// TwinCAT 3 PLC project PLC_Project_XYZ
// ProgramVersion: 3.1.4026.12
// CompilerDefines: VISU_USEPROPERTYINFO
// libraries:
//   Tc2_MC2, * (Beckhoff Automation GmbH)
//   Tc2_Standard, * (Beckhoff Automation GmbH)
//   Tc2_System, * (Beckhoff Automation GmbH)
//   Tc3_Module, * (Beckhoff Automation GmbH)
//   VisuSymbols, 4.5.0.0 (System)
// project tree:
//   / GlobalTextList.TcGTLO, PlcTask.TcTTO, Visualization Manager.TcVMO (not stored)
//   GVLs/ GVL.TcGVL
//   POUs/ MAIN.TcPOU
//   VISUs/ Visu.TcVIS
// real-time tasks:
//   TASK PlcTask: cycle T#10ms, priority 20, ADS port 350
// motion (NC):
//   TASK NC-Task 1 SAF: cycle T#2ms, priority 4, ADS port 501
//   TASK NC-Task 1 SVB: cycle T#10ms, priority 8, ADS port 511
//   AXIS Axis 1 (id 1)
//     OtherSettings: AllowMotionCmdToSlave=true
//     encoder EncType=4
//       EncPara: ScaleFactorNumerator=60, ScaleFactorDenominator=12800, MaxCount=#x0000ffff
//         Inc: RefSoftSyncMask=#x0000ffff
//     drive DrvType=24
//       Analog: VeloReferenz=600, TorqueSetpointScale=10, ScaleFactorActTorque=0.1
//       TimeComp: TaskDelayCycles=1
//     controller CtrType=1
//       CtrPara: PriorControlFactor=1
//         Observer: BandWidth=20
//   AXIS Axis 2 (id 2)
//     OtherSettings: AllowMotionCmdToSlave=true
//     encoder EncType=4
//       EncPara: ScaleFactorNumerator=60, ScaleFactorDenominator=12800, MaxCount=#x0000ffff
//         Inc: RefSoftSyncMask=#x0000ffff
//     drive DrvType=24
//       Analog: VeloReferenz=600, TorqueSetpointScale=10, ScaleFactorActTorque=0.1
//       TimeComp: TaskDelayCycles=1
//     controller CtrType=1
//       CtrPara: PriorControlFactor=1
//         Observer: BandWidth=20
//   AXIS Axis 3 (id 3)
//     OtherSettings: AllowMotionCmdToSlave=true
//     encoder EncType=4
//       EncPara: ScaleFactorNumerator=60, ScaleFactorDenominator=12800, MaxCount=#x0000ffff
//         Inc: RefSoftSyncMask=#x0000ffff
//     drive DrvType=24
//       Analog: VeloReferenz=600, TorqueSetpointScale=10, ScaleFactorActTorque=0.1
//       TimeComp: TaskDelayCycles=1
//     controller CtrType=1
//       CtrPara: PriorControlFactor=1
//         Observer: BandWidth=20
//   AXIS Axis 4 (id 4)
//     OtherSettings: AllowMotionCmdToSlave=true
//     encoder EncType=4
//       EncPara: ScaleFactorNumerator=60, ScaleFactorDenominator=12800, MaxCount=#x0000ffff
//         Inc: RefSoftSyncMask=#x0000ffff
//     drive DrvType=24
//       Analog: VeloReferenz=600, TorqueSetpointScale=10, ScaleFactorActTorque=0.1
//       TimeComp: TaskDelayCycles=1
//     controller CtrType=1
//       CtrPara: PriorControlFactor=1
//         Observer: BandWidth=20
// I/O:
//   DEVICE Device 1 (EtherCAT), AmsNetId 199.4.42.250.2.1
//     Term 1 (EK1200) [EK1200-5000 EtherCAT Power supply (2A E-Bus)]
//       Term 2 (EL1008) [EL1008 8Ch. Dig. Input 24V, 3ms]
//       Term 3 (EL2008) [EL2008 8Ch. Dig. Output 24V, 0.5A]
//       Term 4 (EL3062) [EL3062 2Ch. Ana. Input 0-10V]
//       Term 5 (EL4002) [EL4002 2Ch. Ana. Output 0-10V, 12bit]
//       Term 6 (EK1110) [EK1110 EtherCAT extension]
//     Term 7 (EK1100) [EK1100 EtherCAT Coupler (2A E-Bus)]
//       Term 8 (EL7031-0030) [EL7031-0030 1Ch. Stepper motor output stage (24V, 2.8A)]
//       Term 9 (EL7031-0030) [EL7031-0030 1Ch. Stepper motor output stage (24V, 2.8A)]
//       Term 10 (EL7031-0030) [EL7031-0030 1Ch. Stepper motor output stage (24V, 2.8A)]
//       Term 11 (EL7031-0030) [EL7031-0030 1Ch. Stepper motor output stage (24V, 2.8A)]
//       Term 12 (EL1008) [EL1008 8Ch. Dig. Input 24V, 3ms]
//       Term 13 (EK1110) [EK1110 EtherCAT extension]
//   DEVICE Device 2 (EtherCAT Automation Protocol), AmsNetId 199.4.42.250.3.1
//   DEVICE Device 3 (NOV-DP-RAM)
// variable links:
//   NC-Task 1 SAF/Axes/Axis 1 <-> Device 1 (EtherCAT)/Term 7 (EK1100)/Term 8 (EL7031-0030)
//     Drive/Inputs/In/nState1 @bit 3 <-> STM Status/Status/Error
//     Drive/Inputs/In/nState1 @bit 5 <-> STM Status/Status/Moving negative
//     Drive/Inputs/In/nState1 @bit 4 <-> STM Status/Status/Moving positive
//     Drive/Inputs/In/nState1 @bit 1 <-> STM Status/Status/Ready
//     Drive/Inputs/In/nState1 <-> STM Status/Status/Ready to enable
//     Drive/Inputs/In/nState1 @bit 6 <-> STM Status/Status/Torque reduced
//     Drive/Inputs/In/nState1 @bit 2 <-> STM Status/Status/Warning
//     Drive/Inputs/In/nState2 @bit 3 <-> STM Status/Status/Digital input 1
//     Drive/Inputs/In/nState2 @bit 4 <-> STM Status/Status/Digital input 2
//     Drive/Inputs/In/nState2 @bit 5 <-> STM Status/Status/Sync error
//     Drive/Inputs/In/nState2 @bit 7 <-> STM Status/Status/TxPDO Toggle
//     Drive/Inputs/In/nState4 @bit 1 <-> WcState/InputToggle
//     Drive/Inputs/In/nState4 <-> WcState/WcState
//     Drive/Outputs/Out/nCtrl1 <-> STM Control/Control/Enable
//     Drive/Outputs/Out/nCtrl1 @bit 2 <-> STM Control/Control/Reduce torque
//     Drive/Outputs/Out/nCtrl1 @bit 1 <-> STM Control/Control/Reset
//     Drive/Outputs/Out/nDataOut2[0] <-> STM Velocity/Velocity
//     Enc/Inputs/In/nDataIn1[0] <-> ENC Status compact/Counter value
//     Enc/Inputs/In/nDataIn2[0] <-> ENC Status compact/Latch value
//     Enc/Inputs/In/nState1 @bit 4 <-> ENC Status compact/Status/Counter overflow
//     Enc/Inputs/In/nState1 @bit 3 <-> ENC Status compact/Status/Counter underflow
//     Enc/Inputs/In/nState1 @bit 1 <-> ENC Status compact/Status/Latch extern valid
//     Enc/Inputs/In/nState1 @bit 2 <-> ENC Status compact/Status/Set counter done
//     Enc/Inputs/In/nState2 @bit 4 <-> ENC Status compact/Status/Status of extern latch
//     Enc/Inputs/In/nState2 @bit 5 <-> ENC Status compact/Status/Sync error
//     Enc/Inputs/In/nState2 @bit 7 <-> ENC Status compact/Status/TxPDO Toggle
//     Enc/Inputs/In/nState4 @bit 1 <-> WcState/InputToggle
//     Enc/Inputs/In/nState4 <-> WcState/WcState
//     Enc/Outputs/Out/nCtrl1 @bit 3 <-> ENC Control compact/Control/Enable latch extern on negative edge
//     Enc/Outputs/Out/nCtrl1 @bit 1 <-> ENC Control compact/Control/Enable latch extern on positive edge
//     Enc/Outputs/Out/nCtrl1 @bit 2 <-> ENC Control compact/Control/Set counter
//     Enc/Outputs/Out/nDataOut1[0] <-> ENC Control compact/Set counter value
//   NC-Task 1 SAF/Axes/Axis 2 <-> Device 1 (EtherCAT)/Term 7 (EK1100)/Term 9 (EL7031-0030)
//     Drive/Inputs/In/nState1 @bit 3 <-> STM Status/Status/Error
//     Drive/Inputs/In/nState1 @bit 5 <-> STM Status/Status/Moving negative
//     Drive/Inputs/In/nState1 @bit 4 <-> STM Status/Status/Moving positive
//     Drive/Inputs/In/nState1 @bit 1 <-> STM Status/Status/Ready
//     Drive/Inputs/In/nState1 <-> STM Status/Status/Ready to enable
//     Drive/Inputs/In/nState1 @bit 6 <-> STM Status/Status/Torque reduced
//     Drive/Inputs/In/nState1 @bit 2 <-> STM Status/Status/Warning
//     Drive/Inputs/In/nState2 @bit 3 <-> STM Status/Status/Digital input 1
//     Drive/Inputs/In/nState2 @bit 4 <-> STM Status/Status/Digital input 2
//     Drive/Inputs/In/nState2 @bit 5 <-> STM Status/Status/Sync error
//     Drive/Inputs/In/nState2 @bit 7 <-> STM Status/Status/TxPDO Toggle
//     Drive/Inputs/In/nState4 @bit 1 <-> WcState/InputToggle
//     Drive/Inputs/In/nState4 <-> WcState/WcState
//     Drive/Outputs/Out/nCtrl1 <-> STM Control/Control/Enable
//     Drive/Outputs/Out/nCtrl1 @bit 2 <-> STM Control/Control/Reduce torque
//     Drive/Outputs/Out/nCtrl1 @bit 1 <-> STM Control/Control/Reset
//     Drive/Outputs/Out/nDataOut2[0] <-> STM Velocity/Velocity
//     Enc/Inputs/In/nDataIn1[0] <-> ENC Status compact/Counter value
//     Enc/Inputs/In/nDataIn2[0] <-> ENC Status compact/Latch value
//     Enc/Inputs/In/nState1 @bit 4 <-> ENC Status compact/Status/Counter overflow
//     Enc/Inputs/In/nState1 @bit 3 <-> ENC Status compact/Status/Counter underflow
//     Enc/Inputs/In/nState1 @bit 1 <-> ENC Status compact/Status/Latch extern valid
//     Enc/Inputs/In/nState1 @bit 2 <-> ENC Status compact/Status/Set counter done
//     Enc/Inputs/In/nState2 @bit 4 <-> ENC Status compact/Status/Status of extern latch
//     Enc/Inputs/In/nState2 @bit 5 <-> ENC Status compact/Status/Sync error
//     Enc/Inputs/In/nState2 @bit 7 <-> ENC Status compact/Status/TxPDO Toggle
//     Enc/Inputs/In/nState4 @bit 1 <-> WcState/InputToggle
//     Enc/Inputs/In/nState4 <-> WcState/WcState
//     Enc/Outputs/Out/nCtrl1 @bit 3 <-> ENC Control compact/Control/Enable latch extern on negative edge
//     Enc/Outputs/Out/nCtrl1 @bit 1 <-> ENC Control compact/Control/Enable latch extern on positive edge
//     Enc/Outputs/Out/nCtrl1 @bit 2 <-> ENC Control compact/Control/Set counter
//     Enc/Outputs/Out/nDataOut1[0] <-> ENC Control compact/Set counter value
//   NC-Task 1 SAF/Axes/Axis 3 <-> Device 1 (EtherCAT)/Term 7 (EK1100)/Term 10 (EL7031-0030)
//     Drive/Inputs/In/nState1 @bit 3 <-> STM Status/Status/Error
//     Drive/Inputs/In/nState1 @bit 5 <-> STM Status/Status/Moving negative
//     Drive/Inputs/In/nState1 @bit 4 <-> STM Status/Status/Moving positive
//     Drive/Inputs/In/nState1 @bit 1 <-> STM Status/Status/Ready
//     Drive/Inputs/In/nState1 <-> STM Status/Status/Ready to enable
//     Drive/Inputs/In/nState1 @bit 6 <-> STM Status/Status/Torque reduced
//     Drive/Inputs/In/nState1 @bit 2 <-> STM Status/Status/Warning
//     Drive/Inputs/In/nState2 @bit 3 <-> STM Status/Status/Digital input 1
//     Drive/Inputs/In/nState2 @bit 4 <-> STM Status/Status/Digital input 2
//     Drive/Inputs/In/nState2 @bit 5 <-> STM Status/Status/Sync error
//     Drive/Inputs/In/nState2 @bit 7 <-> STM Status/Status/TxPDO Toggle
//     Drive/Inputs/In/nState4 @bit 1 <-> WcState/InputToggle
//     Drive/Inputs/In/nState4 <-> WcState/WcState
//     Drive/Outputs/Out/nCtrl1 <-> STM Control/Control/Enable
//     Drive/Outputs/Out/nCtrl1 @bit 2 <-> STM Control/Control/Reduce torque
//     Drive/Outputs/Out/nCtrl1 @bit 1 <-> STM Control/Control/Reset
//     Drive/Outputs/Out/nDataOut2[0] <-> STM Velocity/Velocity
//     Enc/Inputs/In/nDataIn1[0] <-> ENC Status compact/Counter value
//     Enc/Inputs/In/nDataIn2[0] <-> ENC Status compact/Latch value
//     Enc/Inputs/In/nState1 @bit 4 <-> ENC Status compact/Status/Counter overflow
//     Enc/Inputs/In/nState1 @bit 3 <-> ENC Status compact/Status/Counter underflow
//     Enc/Inputs/In/nState1 @bit 1 <-> ENC Status compact/Status/Latch extern valid
//     Enc/Inputs/In/nState1 @bit 2 <-> ENC Status compact/Status/Set counter done
//     Enc/Inputs/In/nState2 @bit 4 <-> ENC Status compact/Status/Status of extern latch
//     Enc/Inputs/In/nState2 @bit 5 <-> ENC Status compact/Status/Sync error
//     Enc/Inputs/In/nState2 @bit 7 <-> ENC Status compact/Status/TxPDO Toggle
//     Enc/Inputs/In/nState4 @bit 1 <-> WcState/InputToggle
//     Enc/Inputs/In/nState4 <-> WcState/WcState
//     Enc/Outputs/Out/nCtrl1 @bit 3 <-> ENC Control compact/Control/Enable latch extern on negative edge
//     Enc/Outputs/Out/nCtrl1 @bit 1 <-> ENC Control compact/Control/Enable latch extern on positive edge
//     Enc/Outputs/Out/nCtrl1 @bit 2 <-> ENC Control compact/Control/Set counter
//     Enc/Outputs/Out/nDataOut1[0] <-> ENC Control compact/Set counter value
//   NC-Task 1 SAF/Axes/Axis 4 <-> Device 1 (EtherCAT)/Term 7 (EK1100)/Term 11 (EL7031-0030)
//     Drive/Inputs/In/nState1 @bit 3 <-> STM Status/Status/Error
//     Drive/Inputs/In/nState1 @bit 5 <-> STM Status/Status/Moving negative
//     Drive/Inputs/In/nState1 @bit 4 <-> STM Status/Status/Moving positive
//     Drive/Inputs/In/nState1 @bit 1 <-> STM Status/Status/Ready
//     Drive/Inputs/In/nState1 <-> STM Status/Status/Ready to enable
//     Drive/Inputs/In/nState1 @bit 6 <-> STM Status/Status/Torque reduced
//     Drive/Inputs/In/nState1 @bit 2 <-> STM Status/Status/Warning
//     Drive/Inputs/In/nState2 @bit 3 <-> STM Status/Status/Digital input 1
//     Drive/Inputs/In/nState2 @bit 4 <-> STM Status/Status/Digital input 2
//     Drive/Inputs/In/nState2 @bit 5 <-> STM Status/Status/Sync error
//     Drive/Inputs/In/nState2 @bit 7 <-> STM Status/Status/TxPDO Toggle
//     Drive/Inputs/In/nState4 @bit 1 <-> WcState/InputToggle
//     Drive/Inputs/In/nState4 <-> WcState/WcState
//     Drive/Outputs/Out/nCtrl1 <-> STM Control/Control/Enable
//     Drive/Outputs/Out/nCtrl1 @bit 2 <-> STM Control/Control/Reduce torque
//     Drive/Outputs/Out/nCtrl1 @bit 1 <-> STM Control/Control/Reset
//     Drive/Outputs/Out/nDataOut2[0] <-> STM Velocity/Velocity
//     Enc/Inputs/In/nDataIn1[0] <-> ENC Status compact/Counter value
//     Enc/Inputs/In/nDataIn2[0] <-> ENC Status compact/Latch value
//     Enc/Inputs/In/nState1 @bit 4 <-> ENC Status compact/Status/Counter overflow
//     Enc/Inputs/In/nState1 @bit 3 <-> ENC Status compact/Status/Counter underflow
//     Enc/Inputs/In/nState1 @bit 1 <-> ENC Status compact/Status/Latch extern valid
//     Enc/Inputs/In/nState1 @bit 2 <-> ENC Status compact/Status/Set counter done
//     Enc/Inputs/In/nState2 @bit 4 <-> ENC Status compact/Status/Status of extern latch
//     Enc/Inputs/In/nState2 @bit 5 <-> ENC Status compact/Status/Sync error
//     Enc/Inputs/In/nState2 @bit 7 <-> ENC Status compact/Status/TxPDO Toggle
//     Enc/Inputs/In/nState4 @bit 1 <-> WcState/InputToggle
//     Enc/Inputs/In/nState4 <-> WcState/WcState
//     Enc/Outputs/Out/nCtrl1 @bit 3 <-> ENC Control compact/Control/Enable latch extern on negative edge
//     Enc/Outputs/Out/nCtrl1 @bit 1 <-> ENC Control compact/Control/Enable latch extern on positive edge
//     Enc/Outputs/Out/nCtrl1 @bit 2 <-> ENC Control compact/Control/Set counter
//     Enc/Outputs/Out/nDataOut1[0] <-> ENC Control compact/Set counter value
//   PLC_Project_XYZ/PLC_Project_XYZ Instance <-> Device 1 (EtherCAT)/Term 1 (EK1200)/Term 2 (EL1008)
//     PlcTask Inputs/MAIN.BTN_LEFT <-> Channel 1/Input
//     PlcTask Inputs/MAIN.BTN_LEFT_B <-> Channel 3/Input
//     PlcTask Inputs/MAIN.BTN_RIGHT <-> Channel 2/Input
//     PlcTask Inputs/MAIN.BTN_RIGHT_B <-> Channel 4/Input
//   PLC_Project_XYZ/PLC_Project_XYZ Instance <-> Device 1 (EtherCAT)/Term 1 (EK1200)/Term 4 (EL3062)
//     PlcTask Inputs/MAIN.nPotentiometer <-> AI Standard Channel 1/Value
//   PLC_Project_XYZ/PLC_Project_XYZ Instance <-> Device 1 (EtherCAT)/Term 7 (EK1100)/Term 12 (EL1008)
//     PlcTask Inputs/MAIN.SWX1 <-> Channel 2/Input
//     PlcTask Inputs/MAIN.SWX2 <-> Channel 1/Input
//     PlcTask Inputs/MAIN.SWY1 <-> Channel 3/Input
//     PlcTask Inputs/MAIN.SWY2 <-> Channel 4/Input
//   PLC_Project_XYZ/PLC_Project_XYZ Instance <-> NC-Task 1 SAF/Axes/Axis 1
//     PlcTask Inputs/MAIN.Axis_y1.NcToPlc <-> Outputs/ToPlc
//     PlcTask Outputs/MAIN.Axis_y1.PlcToNc <-> Inputs/FromPlc
//   PLC_Project_XYZ/PLC_Project_XYZ Instance <-> NC-Task 1 SAF/Axes/Axis 2
//     PlcTask Inputs/MAIN.Axis_y2.NcToPlc <-> Outputs/ToPlc
//     PlcTask Outputs/MAIN.Axis_y2.PlcToNc <-> Inputs/FromPlc
//   PLC_Project_XYZ/PLC_Project_XYZ Instance <-> NC-Task 1 SAF/Axes/Axis 3
//     PlcTask Inputs/MAIN.Axis_z.NcToPlc <-> Outputs/ToPlc
//     PlcTask Outputs/MAIN.Axis_z.PlcToNc <-> Inputs/FromPlc
//   PLC_Project_XYZ/PLC_Project_XYZ Instance <-> NC-Task 1 SAF/Axes/Axis 4
//     PlcTask Inputs/MAIN.Axis_x.NcToPlc <-> Outputs/ToPlc
//     PlcTask Outputs/MAIN.Axis_x.PlcToNc <-> Inputs/FromPlc

CONFIGURATION PLC_Project_XYZ
    RESOURCE PLC ON TwinCAT3
        TASK PlcTask(INTERVAL := T#10ms, PRIORITY := 20);
        PROGRAM MAIN WITH PlcTask : MAIN;
    END_RESOURCE
END_CONFIGURATION

// ---- GVLs/GVL.TcGVL
{attribute 'qualified_only'}
VAR_GLOBAL
	//Leds
	bLed_Rd1 AT %Q* : BOOL;
	bLed_Rd2 AT %Q* : BOOL;
	bLed_Rd3 AT %Q* : BOOL;
	bLed_Rd4 AT %Q* : BOOL;
	
	bLed_Gn1 AT %Q* : BOOL;
	bLed_Gn2 AT %Q* : BOOL;
	bLed_Gn3 AT %Q* : BOOL;
	bLed_Gn4 AT %Q* : BOOL;
	
	//Buttons
	bButton1 	AT %I* : BOOL;
    bButton2 	AT %I* : BOOL;
    bButton3 	AT %I* : BOOL;
    bButton4 	AT %I* : BOOL;
	bButton5 	AT %I* : BOOL;
    bButton6 	AT %I* : BOOL;
	bHome 		AT %I* : BOOL;
	
	//Sliders
	slider1 : INT;
	slider2 : INT;
	slider3 : INT;
END_VAR

// ---- POUs/MAIN.TcPOU
PROGRAM MAIN
VAR

	START : BOOL := FALSE;

    // input
	bJogF	: BOOL := FALSE;
	bJogB	: BOOL := FALSE;
	bSet 	: BOOL := FALSE;
	bToggle : BOOL := FALSE;
	nValue AT %I*: LREAL;
    nPotentiometer AT %I*: INT;
    nDisplay AT %Q*: INT;
	
	
    ExecuteABS        : BOOL;
    Enable          : BOOL := TRUE;
    Enable_Positive : BOOL := TRUE;
    Enable_Negative : BOOL := TRUE;
    Override        : LREAL := 100.0;
    BufferMode      : MC_BufferMode;
    Options         : ST_PowerOptions;
    BTN_RIGHT       AT %I* : BOOL := FALSE;
    BTN_LEFT        AT %I* : BOOL := FALSE;

	BTN_RIGHT_B		AT %I* : BOOL := FALSE;
	BTN_LEFT_B		AT %I* : BOOL := FALSE;
	
    SWY1  AT %I* : BOOL;
    SWY2  AT %I* : BOOL;
    SWX1  AT %I* : BOOL;
    SWX2  AT %I* : BOOL;

    // output
    Status  : BOOL;
    Busy    : BOOL;
    Active  : BOOL;
    Error   : BOOL;
    ErrorID : UDINT;



	



    Axis_x : AXIS_REF;
	Axis_z : AXIS_REF;
	
	Axis_y1 : AXIS_REF;
	Axis_y2 : AXIS_REF;
	
	

    mc_power : MC_Power;
	mc_powerZ : MC_Power;
	mc_powerY1: MC_Power;
	mc_powerY2: MC_Power;

    fbMoveAbsX1: MC_MoveAbsolute;
    fbMoveAbsX2: MC_MoveAbsolute;
	fbMoveAbsY1: MC_MoveAbsolute;
    fbMoveAbsY2: MC_MoveAbsolute;
	fbMoveAbsZ1: MC_MoveAbsolute;
    fbMoveAbsZ2: MC_MoveAbsolute;
	

	Axis_x_Halt: MC_Halt;
	Halt_X1: MC_Halt;
	Halt_X2: MC_Halt;
	
	Axis_y_Halt: MC_Halt;
	Halt_Y1: MC_Halt;
	Halt_Y2: MC_Halt;
	
	Axis_z_Halt: MC_Halt;
	Halt_Z1: MC_Halt;
	Halt_Z2: MC_Halt;
	
	
	Couple_Y1_Y2: MC_GearInDyn;
	fb_Jog_Z: MC_Jog;
	fb_Jog_X: MC_Jog;
	fb_Jog_Y: MC_Jog;
	
END_VAR

mc_power.Enable := Enable;
mc_powerZ.Enable := Enable;
mc_powerY1.Enable:= Enable;
mc_powerY2.Enable:= Enable;

mc_power.Enable_Positive := Enable_Positive;
mc_power.Enable_Negative := Enable_Negative;
mc_power.Override := Override;

mc_powerZ.Enable_Positive := Enable_Positive;
mc_powerZ.Enable_Negative := Enable_Negative;
mc_powerZ.Override := Override;

mc_powerY1.Enable_Positive := Enable_Positive;
mc_powerY1.Enable_Negative := Enable_Negative;
mc_powerY1.Override := Override;

mc_powerY2.Enable_Positive := Enable_Positive;
mc_powerY2.Enable_Negative := Enable_Negative;
mc_powerY2.Override := Override;

mc_power(Axis := Axis_x );
mc_powerZ(Axis := Axis_z );
mc_powerY1(Axis := Axis_y1 );
mc_powerY2(Axis := Axis_y2 );


Couple_Y1_Y2(
	Master:= Axis_y1, 
	Slave:= Axis_y2, 
	Enable:= TRUE, 
	GearRatio:= 1, 
	Acceleration:= , 
	Deceleration:= , 
	Jerk:= , 
	BufferMode:= , 
	Options:= , 
	InGear=> , 
	Busy=> , 
	Active=> , 
	CommandAborted=> , 
	Error=> , 
	ErrorID=> );

fbMoveAbsX1(
	Axis        := Axis_x, 
	Execute     := (START OR gvl.bHome) AND NOT SWX1, 
	Position    := gvl.slider1, 
	Velocity    := 50, 

);


	
//fbMoveAbsX2(
//    Axis        := Axis_x, 
//    Execute     := BTN_RIGHT AND NOT SWX2, 
//    Position    := -3000, 
//    Velocity    := 50, 

//    );
Halt_X1(
	Axis:= Axis_x, 
	Execute:= SWX1, 
	 );
	 
//Halt_X2(
//	Axis:= Axis_x, 
//	Execute:= SWX2, 
//	 );
	 

//fbMoveAbsY1(
//    Axis        := Axis_y1, 
//    Execute     := BTN_LEFT_B AND NOT SWY1, 
//    Position    := 3000, 
//    Velocity    := 50, 

//    );
	
fbMoveAbsY2(
    Axis        := Axis_y1, 
    Execute     := (START OR gvl.bHome) AND NOT SWY2, 
    Position    := gvl.slider2, 
    Velocity    := 50, 

    );
//Halt_Y1(
//	Axis:= Axis_y1, 
//	Execute:= SWY1, 
//	 );
	 
Halt_Y2(
	Axis:= Axis_y1, 
	Execute:= SWY2, 
	 );

nValue := TO_INT (nPotentiometer*1000/32767);
IF(nValue < 100 ) THEN
	bJogF := TRUE;
	bJogB := FALSE;
ELSIF(nValue > 300) THEN
	bJogB := TRUE;
	bJogF := FALSE;
ELSE
	bJogB := FALSE;
	bJogF := FALSE;
END_IF

	 
fb_Jog_Z(
	Axis:= Axis_z, 
	JogForward:= bJogF OR gvl.bButton6, 
	JogBackwards:= bJogB OR gvl.bButton5, 
	Mode:= , 
	Position:= , 
	Velocity:= 50, 
	Acceleration:= , 
	Deceleration:= , 
	Jerk:= , 
	Done=> , 
	Busy=> , 
	Active=> , 
	CommandAborted=> , 
	Error=> , 
	ErrorID=> );

fb_Jog_y(
	Axis:= Axis_y1, 
	JogForward:= (BTN_RIGHT_B OR gvl.bButton4) AND NOT SWY1, 
	JogBackwards:= (BTN_LEFT_B OR gvl.bButton3) AND NOT SWY2, 
	Mode:= , 
	Position:= , 
	Velocity:= 50, 
	Acceleration:= , 
	Deceleration:= , 
	Jerk:= , 
	Done=> , 
	Busy=> , 
	Active=> , 
	CommandAborted=> , 
	Error=> , 
	ErrorID=> );
	
fb_Jog_X(
	Axis:= Axis_x, 
	JogForward:= (BTN_RIGHT OR gvl.bButton2) AND NOT SWX1, 
	JogBackwards:= (BTN_LEFT OR gvl.bButton1) AND NOT SWX2, 
	Mode:= , 
	Position:= , 
	Velocity:= 50, 
	Acceleration:= , 
	Deceleration:= , 
	Jerk:= , 
	Done=> , 
	Busy=> , 
	Active=> , 
	CommandAborted=> , 
	Error=> , 
	ErrorID=> );
	
GVL.bLed_Gn1 := Axis_x.Status.ControlLoopClosed;
gvl.bLed_Rd1 := Axis_x.Status.Error;
GVL.bLed_Gn2 := Axis_y1.Status.ControlLoopClosed;
gvl.bLed_Rd2 := Axis_y1.Status.Error;
GVL.bLed_Gn3 := Axis_y2.Status.ControlLoopClosed;
gvl.bLed_Rd3 := Axis_y2.Status.Error;
GVL.bLed_Gn4 := Axis_z.Status.ControlLoopClosed;
gvl.bLed_Rd4 := Axis_z.Status.Error;

END_PROGRAM

// ---- GlobalTextList.TcGTLO
TEXTLIST GlobalTextList
  237 = '+'
  569 = '-'
  720 = 'Axes Status'
  276 = 'Button 1'
  310 = 'Control Panel'
  422 = 'Home Panel'
  355 = 'X Axes'
  817 = 'X Axis'
  545 = 'Y Axes'
  114 = 'Y1 Axis'
  398 = 'Y2 Axis'
  842 = 'Z Axes'
  294 = 'Z Axis'
END_TEXTLIST

// ---- VISUs/Visu.TcVIS
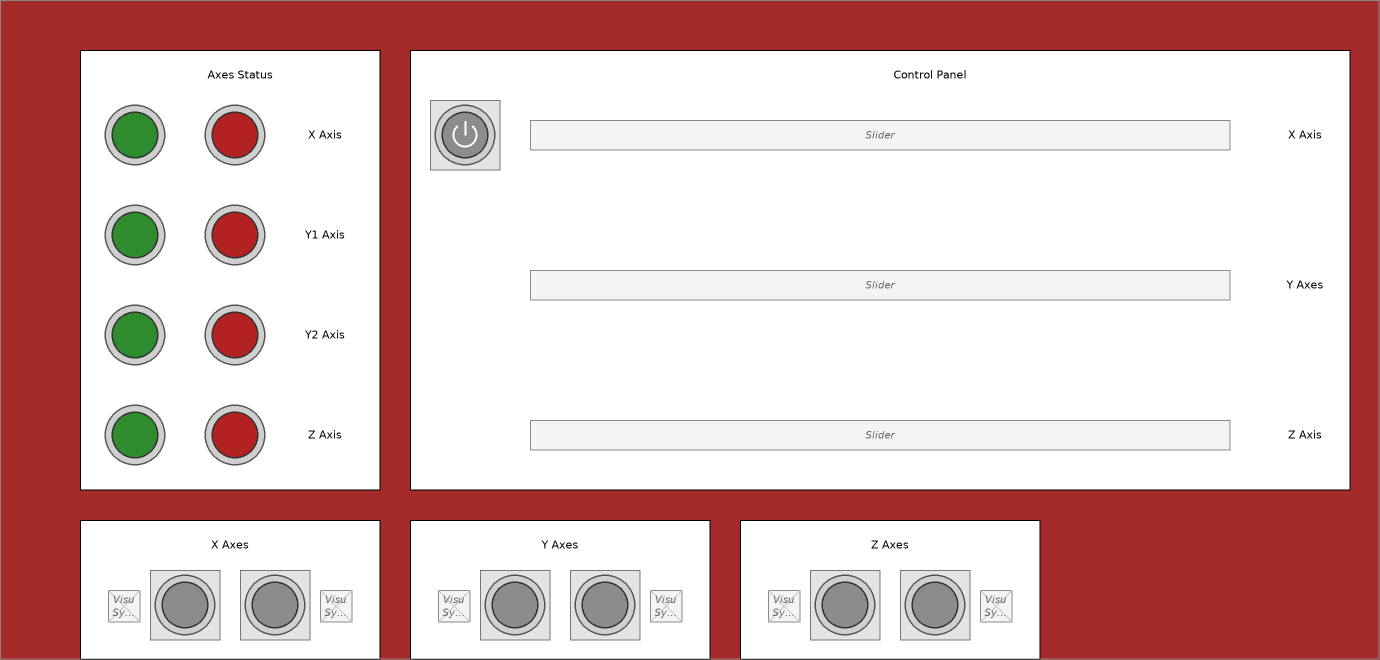
VISUALIZATION Visu  // 1380x660
    Rectangle (80,50 300x440)
    Lamp1 (100,100 70x70), variable: GVL.bLed_Gn1, style: Lamp-Lamp1-Green
    Lamp1 (100,200 70x70), variable: GVL.bLed_Gn2, style: Lamp-Lamp1-Green
    Lamp1 (100,300 70x70), variable: GVL.bLed_Gn3, style: Lamp-Lamp1-Green
    Lamp1 (100,400 70x70), variable: GVL.bLed_Gn4, style: Lamp-Lamp1-Green
    Label (165,60 150x30), "Axes Status"
    Lamp1 (200,100 70x70), variable: GVL.bLed_Rd1, style: Lamp-Lamp1-Red
    Lamp1 (200,200 70x70), variable: GVL.bLed_Rd2, style: Lamp-Lamp1-Red
    Lamp1 (200,300 70x70), variable: GVL.bLed_Rd3, style: Lamp-Lamp1-Red
    Lamp1 (200,400 70x70), variable: GVL.bLed_Rd4, style: Lamp-Lamp1-Red
    Label (250,120 150x30), "X Axis"
    Label (250,220 150x30), "Y1 Axis"
    Label (250,320 150x30), "Y2 Axis"
    Label (250,420 150x30), "Z Axis"
    Rectangle (410,50 940x440)
    Slider (530,120 700x30), variable: GVL.slider1, scale 0..375
    Slider (530,270 700x30), variable: GVL.slider2, scale 0..375
    Slider (530,420 700x30), variable: GVL.slider3, scale 0..125
    Label (855,60 150x30), "Control Panel"
    Label (1230,420 150x30), "Z Axis"
    Label (1230,270 150x30), "Y Axes"
    Label (1230,120 150x30), "X Axis"
    Rectangle (80,520 300x140)
    PushSwitch (150,570 70x70), variable: GVL.bButton1, behaviour: TOGGLE, style: Switch-PushSwitch-Gray
    PushSwitch (240,570 70x70), variable: GVL.bButton2, behaviour: TOGGLE, style: Switch-PushSwitch-Gray
    Label (155,530 150x30), "X Axes"
    Label (620,590 150x30), "+"
    Rectangle (410,520 300x140)
    PushSwitch (480,570 70x70), variable: GVL.bButton3, behaviour: TOGGLE, style: Switch-PushSwitch-Gray
    PushSwitch (570,570 70x70), variable: GVL.bButton4, behaviour: TOGGLE, style: Switch-PushSwitch-Gray
    Label (485,530 150x30), "Y Axes"
    Rectangle (740,520 300x140)
    PushSwitch (810,570 70x70), variable: GVL.bButton5, behaviour: TOGGLE, style: Switch-PushSwitch-Gray
    PushSwitch (900,570 70x70), variable: GVL.bButton6, behaviour: TOGGLE, style: Switch-PushSwitch-Gray
    Label (815,530 150x30), "Z Axes"
    Image (320,590 32x32), image: VisuSymbols.Symbols.ArrowBoldRight
    Image (650,590 32x32), image: VisuSymbols.Symbols.ArrowBoldRight
    Image (980,590 32x32), image: VisuSymbols.Symbols.ArrowBoldRight
    Image (108,590 32x32), image: VisuSymbols.Symbols.ArrowBoldLeft
    Image (438,590 32x32), image: VisuSymbols.Symbols.ArrowBoldLeft
    Image (768,590 32x32), image: VisuSymbols.Symbols.ArrowBoldLeft
    PowerSwitch (430,100 70x70), variable: GVL.bHome, behaviour: TAP, style: Switch-PowerSwitch-Gray
END_VISUALIZATION
